FUNCTION_BLOCK AE2_TO_AE (* Composite FB for convert bidirectional AE2 to unidirectional AE *)
  (* Standard: 61499-2; Function: AE2_BIDIR forwards its incoming (EO1) side out as a plain unidirectional event via AE_OUT. AE_IN publishes its event onto the outgoing (EI1) side of AE2_BIDIR.; Description: Copyright (c) 2026 HR Agrartechnik GmbH This program and the accompanying materials are made available under the terms of the Eclipse Public License 2.0 which is available at https://www.eclipse.org/legal/epl-2.0/ SPDX-License-Identifier: EPL-2.0 *)
  (* Version 1.0, 2026-08-31, Franz Höpfinger, HR Agrartechnik GmbH, Initial Version *)
  PACKAGE adapter::conversion::bidirectional;
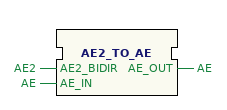
  SOCKETS
    AE2_BIDIR : adapter::types::bidirectional::AE2; (* Adapter Input: bidirectional tap, incoming side forwarded to AE_OUT, outgoing side driven by AE_IN *)
    AE_IN : adapter::types::unidirectional::AE; (* Adapter Input: unidirectional source *)
  END_SOCKETS
  PLUGS
    AE_OUT : adapter::types::unidirectional::AE; (* Adapter Output: mirrors AE2_BIDIR's incoming (indication) side *)
  END_PLUGS
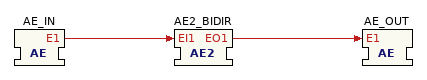
  EVENT_CONNECTIONS
    AE2_BIDIR.EO1 TO AE_OUT.E1;
    AE_IN.E1 TO AE2_BIDIR.EI1;
  END_CONNECTIONS
END_FUNCTION_BLOCK
